(* IEC 61131-3 sources: Std_PalletMover/Class/PL221 (part 2) *)

//https://jonasjacek.github.io/colors/

END_FUNCTION

FUNCTION VIRTUAL PL221::IndividualStripeConfig

//Example for Stripe Type WS2813

//  IndividualStripeCon1.PixelOrder      := GRB;
//  IndividualStripeCon1.LSBFirstOut     := FALSE; // BOOL
//  IndividualStripeCon1.PixelOutT0H     := 400;   //value in ns
//  IndividualStripeCon1.PixelOutT1H     := 900;   //value in ns
//  IndividualStripeCon1.PixelOutT0L     := 800;   //value in ns
//  IndividualStripeCon1.PixelOutT1L     := 800;   //value in ns
//  IndividualStripeCon1.ResetPixelTime  := 310;   //value in ns

END_FUNCTION
